// TIA Portal V17 export
// export: Created 2023-12-22T15:05:29.6970183Z, ExportSetting WithDefaults, DisplayName Totally Integrated Automation Portal, DisplayVersion V17, DisplayName TIA Portal Openness, DisplayVersion V17, DisplayName TIA Portal Version Control Interface, DisplayVersion V17, DisplayName STEP 7 Professional, DisplayVersion V17, DisplayName STEP 7 Safety, DisplayVersion V17, DisplayName WinCC Advanced, DisplayVersion V17
DATA_BLOCK "AOx_DB"   // DB230
VERSION : 0.1
// stored: AutoNumber false, DBAccessibleFromOPCUA true, InstanceOfName AOx, InstanceOfType FB
"AOx"
   // VAR RETAIN
   //    Time_DTL { S7_SetPoint := 'True'} : DTL := DTL#2012-01-01-20:29:23.453503;
   // END_VAR
BEGIN
END_DATA_BLOCK
